// TIA Portal V16 export
// export: Created 2021-11-12T13:32:46.4783866Z, ExportSetting WithDefaults, DisplayName Totally Integrated Automation Portal, DisplayVersion V16 Update 3, DisplayName TIA Portal Version Control Interface, DisplayVersion V16 Update 2, DisplayName TIA Portal Openness, DisplayVersion V16 Update 3, DisplayName SINAMICS Startdrive Advanced, DisplayVersion V16 Update 5, DisplayName SINAMICS Startdrive G130, G150, S120, S150, SINAMICS MV, S210, DisplayVersion V16 Update 5, DisplayName SINAMICS Startdrive G110M, G120, G120C, G120D, G120P, G115D, DisplayVersion V16 Update 5, DisplayName STEP 7 Professional, DisplayVersion V16 Update 3, DisplayName STEP 7 Safety, DisplayVersion V16, DisplayName WinCC UA Professional, DisplayVersion V16 Update 3
DATA_BLOCK "STATUS_Zone200"   // DB25
{ S7_Optimized_Access := 'TRUE'; DB_Accessible_From_OPC_UA := 'FALSE' }
VERSION : 0.1
// stored: AutoNumber true, DBAccessibleFromOPCUA false, IsOnlyStoredInLoadMemory false, IsRetainMemResEnabled false, IsWriteProtectedInAS false, MemoryReserve 100
   VAR
      Mode : Struct   // Statuses and error of zone 200
         Main : "UDT_Status_main";
         Specific : "UDT_Zone_Status_specific";
         Error : "UDT_Error01";
      END_STRUCT;
      Station210_Mode : Struct   // Statuses and error of station 210
         Main : "UDT_Status_main";
         Specific : "UDT_Zone_Status_specific";
         Error : "UDT_Error01";
      END_STRUCT;
      Station220_Mode : Struct   // Statuses and error of station 220
         Main : "UDT_Status_main";
         Specific : "UDT_Zone_Status_specific";
         Error : "UDT_Error01";
      END_STRUCT;
      Station230_Mode : Struct   // Statuses and error of station 230
         Main : "UDT_Status_main";
         Specific : "UDT_Zone_Status_specific";
         Error : "UDT_Error01";
      END_STRUCT;
      Station2R1_Mode : Struct   // Statuses and error of station 2R1
         Main : "UDT_Status_main";
         Specific : "UDT_Zone_Status_specific";
         Error : "UDT_Error01";
      END_STRUCT;
      Station2R2_Mode : Struct   // Statuses and error of station 2R2
         Main : "UDT_Status_main";
         Specific : "UDT_Zone_Status_specific";
         Error : "UDT_Error01";
      END_STRUCT;
      StationSCH1_Mode : Struct   // Statuses and error of station SCH1
         Main : "UDT_Status_main";
         Specific : "UDT_Zone_Status_specific";
         Error : "UDT_Error01";
      END_STRUCT;
      StationBSN3_Mode : Struct   // Statuses and error of station BSN3
         Main : "UDT_Status_main";
         Specific : "UDT_Zone_Status_specific";
         Error : "UDT_Error01";
      END_STRUCT;
      "RU01-KF02" : Struct   // Status of bus module RU01-KF01
         Main : "UDT_Status_main";
         Specific { S7_SetPoint := 'True'} : "UDT_EuchnerSafetySwitch2MBM_Status_Specific";
         Error { S7_SetPoint := 'True'} : "UDT_Error01";
      END_STRUCT;
      "RU01-KF03" : Struct   // Status of bus module RU01-KF01
         Main : "UDT_Status_main";
         Specific { S7_SetPoint := 'True'} : "UDT_EuchnerSafetySwitch2MBM_Status_Specific";
         Error { S7_SetPoint := 'True'} : "UDT_Error01";
      END_STRUCT;
      "RU01-KF04" : Struct   // Status of bus module RU01-KF01
         Main : "UDT_Status_main";
         Specific { S7_SetPoint := 'True'} : "UDT_EuchnerSafetySwitch2MBM_Status_Specific";
         Error { S7_SetPoint := 'True'} : "UDT_Error01";
      END_STRUCT;
      "RU01-QQ01" : Struct   // Status of gate 100+RU01-QQ01
         Main : "UDT_Status_main";
         Specific { S7_SetPoint := 'True'} : "UDT_Door_MGB2_L1_Status_specific";
         Error { S7_SetPoint := 'True'} : "UDT_Error01";
      END_STRUCT;
      "RU01-QQ02" : Struct   // Status of gate 100+RU01-QQ02
         Main : "UDT_Status_main";
         Specific { S7_SetPoint := 'True'} : "UDT_Door_MGB2_L1_Status_specific";
         Error { S7_SetPoint := 'True'} : "UDT_Error01";
      END_STRUCT;
      "RU01-QQ03" : Struct   // Status of gate 100+RU01-QQ03
         Main : "UDT_Status_main";
         Specific { S7_SetPoint := 'True'} : "UDT_Door_MGB2_L1_Status_specific";
         Error { S7_SetPoint := 'True'} : "UDT_Error01";
      END_STRUCT;
      "RU01-QQ04" : Struct   // Status of gate 100+RU01-QQ04
         Main : "UDT_Status_main";
         Specific { S7_SetPoint := 'True'} : "UDT_Door_MGB2_L1_Status_specific";
         Error { S7_SetPoint := 'True'} : "UDT_Error01";
      END_STRUCT;
      "RU01-QQ05" : Struct   // Status of gate 100+RU01-QQ05
         Main : "UDT_Status_main";
         Specific { S7_SetPoint := 'True'} : "UDT_Door_MGB2_L1_Status_specific";
         Error { S7_SetPoint := 'True'} : "UDT_Error01";
      END_STRUCT;
      xxxxx_Alarms__xxxxx : Byte;
      "UF01-SF01" : Struct   // E-stop 200UF01-SF01
         Main { S7_SetPoint := 'True'} : "UDT_Status_main";
         Specific { S7_SetPoint := 'True'} : "UDT_DI_Mon_Status_specific";
         Error { S7_SetPoint := 'True'} : "UDT_Error01";
      END_STRUCT;
      "RU01-QQ01_ES" : Struct   // E-stop gate 200QQ01 / E-stop branka 200QQ01
         Main { S7_SetPoint := 'True'} : "UDT_Status_main";
         Specific { S7_SetPoint := 'True'} : "UDT_DI_Mon_Status_specific";
         Error { S7_SetPoint := 'True'} : "UDT_Error01";
      END_STRUCT;
      "RU01-QQ02_ES" : Struct   // E-stop gate 200QQ02 / E-stop branka 200QQ02
         Main { S7_SetPoint := 'True'} : "UDT_Status_main";
         Specific { S7_SetPoint := 'True'} : "UDT_DI_Mon_Status_specific";
         Error { S7_SetPoint := 'True'} : "UDT_Error01";
      END_STRUCT;
      "RU01-QQ03_ES" : Struct   // E-stop gate 200QQ03 / E-stop branka 200QQ03
         Main { S7_SetPoint := 'True'} : "UDT_Status_main";
         Specific { S7_SetPoint := 'True'} : "UDT_DI_Mon_Status_specific";
         Error { S7_SetPoint := 'True'} : "UDT_Error01";
      END_STRUCT;
      "RU01-QQ04_ES" : Struct   // E-stop gate 200QQ04 / E-stop branka 200QQ04
         Main { S7_SetPoint := 'True'} : "UDT_Status_main";
         Specific { S7_SetPoint := 'True'} : "UDT_DI_Mon_Status_specific";
         Error { S7_SetPoint := 'True'} : "UDT_Error01";
      END_STRUCT;
      "RU01-QQ05_ES" : Struct   // E-stop gate 200QQ05 / E-stop branka 200QQ05
         Main { S7_SetPoint := 'True'} : "UDT_Status_main";
         Specific { S7_SetPoint := 'True'} : "UDT_DI_Mon_Status_specific";
         Error { S7_SetPoint := 'True'} : "UDT_Error01";
      END_STRUCT;
      "RU01-KF2" : Struct   // Gate module 200RU01-KF01 / Modul branky 200RU01-KF01
         Main { S7_SetPoint := 'True'} : "UDT_Status_main";
         Specific { S7_SetPoint := 'True'} : "UDT_DI_Mon_Status_specific";
         Error { S7_SetPoint := 'True'} : "UDT_Error01";
      END_STRUCT;
      "RU01-KF3" : Struct   // Gate module 200RU01-KF02 / Modul branky 200RU01-KF02
         Main { S7_SetPoint := 'True'} : "UDT_Status_main";
         Specific { S7_SetPoint := 'True'} : "UDT_DI_Mon_Status_specific";
         Error { S7_SetPoint := 'True'} : "UDT_Error01";
      END_STRUCT;
      "RU01-KF4" : Struct   // Gate module 200RU01-KF03 / Modul branky 200RU01-KF03
         Main { S7_SetPoint := 'True'} : "UDT_Status_main";
         Specific { S7_SetPoint := 'True'} : "UDT_DI_Mon_Status_specific";
         Error { S7_SetPoint := 'True'} : "UDT_Error01";
      END_STRUCT;
      "RU01-KF5" : Struct   // Gate module 200RU01-KF04 / Modul branky 200RU01-KF04
         Main { S7_SetPoint := 'True'} : "UDT_Status_main";
         Specific { S7_SetPoint := 'True'} : "UDT_DI_Mon_Status_specific";
         Error { S7_SetPoint := 'True'} : "UDT_Error01";
      END_STRUCT;
   END_VAR
BEGIN
END_DATA_BLOCK
